(* PLC project my_app_1, Dassault Systèmes ControlBuild 2024x Refresh1 *)
(* stored: creationDateTime 2024-03-13T18:06:36-01:00 *)

PROGRAM sub1
  VAR_INPUT
    entree : BOOL := false;
    entree2 : BOOL := false;
    entree3 : BOOL := false;
    entree4 : BOOL := false;
  END_VAR

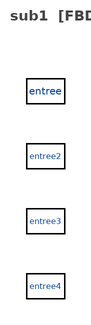
(* FBD diagram, written out as Structured Text *)
(* drawn but not wired to any output: entree, entree2, entree3, entree4 *)
END_PROGRAM

PROGRAM my_app.my_app_1
  VAR_INPUT
    entree : BOOL := false;
  END_VAR

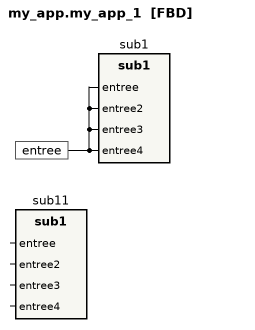
(* FBD diagram, written out as Structured Text *)
sub1(entree := entree, entree2 := entree, entree3 := entree, entree4 := entree);
sub11();
END_PROGRAM
